// TIA Portal V20 export
FUNCTION_BLOCK "CallGlobal"   // FB48, LAD
TITLE = CallGlobal
// All blocks that provide data to the DB Global.Data are called here. That includes blocks to generate system data as well as blocks that connect handle multiple HMIs.
// stored: IsIECCheckEnabled true, MemoryReserve 100, SetENOAutomatically true
   VAR
      statClockSysMemOld { ExternalWritable := 'False'} : Byte;   // Old value system memory evaluation
      statRev0Hz5 : Bool;
      statTonTimer : Array[0..1] of IEC_TIMER;
      instLAF_PowerOnOff { ExternalWritable := 'False'} : "LAF_PowerOnOff";
      instLAF_HmiHeaderManager { ExternalWritable := 'False'} : "LAF_HmiHeaderManager";
      instLAF_ClockGen { ExternalWritable := 'False'} : "LAF_ClockGenerator";
      instLSNTP_Server { ExternalWritable := 'False'} : "LSNTP_Server";
      instRemoteAccess { ExternalWritable := 'False'} : "LRemoteAccess_MobilePanelMonitor";
      statPulse : Array[0..99] of Bool;
   END_VAR
   VAR_TEMP
      tempIndex : DInt;   // Temp variable for for loop
      tempAcknowledge : Bool;   // Summarized acknowledge command
      tempPowerOff : Bool;   // Summarized power off command
      tempPowerOn : Bool;   // Summarized power on command
      tempPowerStatus : Int;   // 0 - Off, 1 - Paused, 2 - On
      tempResultXor : Byte;   // Interim result of XOR operation
      tempPosPulse : Byte;   // Interim result puls calculation
   END_VAR
   VAR CONSTANT
      RESET_BUTTON__COULD_BE_ADDED_HERE : Bool := false;   // Placeholder for a potential global reset button
      TRUE : Bool := true;
      FALSE : Bool;
   END_VAR
   VAR_TEMP   // added for the SCL form of the ladder/FBD networks
      _w1 : Bool;
      _w2 : Bool;
      _w3 : Bool;
      _w4 : Bool;
   END_VAR
BEGIN

REGION Network 1 (SCL): Summarize HMI commands
   // Read commands for acknowledge, powerOn and powerOff from the different HMI panels and summarize them in temp variables for further logic in this block.
   // Initialize temp variables
   #tempAcknowledge :=
   #tempPowerOff :=
   #tempPowerOn := FALSE;

   // Loop through the HMI panels and summarize the commands
   FOR #tempIndex := 0 TO "NO_OF_PANELS" DO
       #tempAcknowledge := #tempAcknowledge OR "Hmi".mainHeader[#tempIndex].hmiToPlc.acknowledge;
       #tempPowerOff := #tempPowerOff OR "Hmi".mainHeader[#tempIndex].hmiToPlc.powerCommands.%X0;
       #tempPowerOn := #tempPowerOn OR "Hmi".mainHeader[#tempIndex].hmiToPlc.powerCommands.%X1;
   END_FOR;
END_REGION

REGION Network 2: Global Acknowledge
   // The global acknowledge command from the hmi button is assigned to Global.Data.general.acknowledge: This bit it forwarded to all underlaying modules
   // If a hard-wired global reset button exists, it can
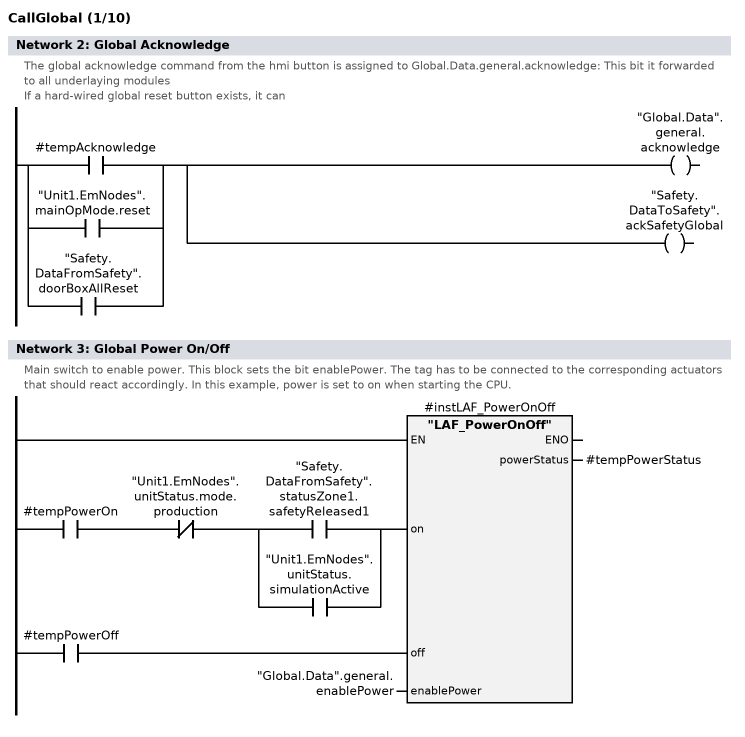
   RUNG wire#powerrail
      Contact( #tempAcknowledge )
      wire#w1
      Coil( "Global.Data".general.acknowledge )
   END_RUNG
   RUNG wire#powerrail
      Contact( "Unit1.EmNodes".mainOpMode.reset )
   END_RUNG wire#w1
   RUNG wire#powerrail
      Contact( "Safety.DataFromSafety".doorBoxAllReset )
   END_RUNG wire#w1
   RUNG wire#w1
      Coil( "Safety.DataToSafety".ackSafetyGlobal )
   END_RUNG
   // the same network as SCL:
   "Global.Data".general.acknowledge := #tempAcknowledge OR "Unit1.EmNodes".mainOpMode.reset OR "Safety.DataFromSafety".doorBoxAllReset;
   "Safety.DataToSafety".ackSafetyGlobal := "Global.Data".general.acknowledge;
END_REGION

REGION Network 3: Global Power On/Off
   // Main switch to enable power. This block sets the bit enablePower. The tag has to be connected to the corresponding actuators that should react accordingly. In this example, power is set to on when starting the CPU.
   RUNG wire#powerrail
      #instLAF_PowerOnOff(on := wire#w2, off := wire#w3, enablePower := "Global.Data".general.enablePower, powerStatus => #tempPowerStatus)
   END_RUNG
   RUNG wire#powerrail
      Contact( #tempPowerOn )
      I_Contact( "Unit1.EmNodes".unitStatus.mode.production )
      wire#w1
      Contact( "Safety.DataFromSafety".statusZone1.safetyReleased1 )
   END_RUNG wire#w2
   RUNG wire#w1
      Contact( "Unit1.EmNodes".unitStatus.simulationActive )
   END_RUNG wire#w2
   RUNG wire#powerrail
      Contact( #tempPowerOff )
   END_RUNG wire#w3
   // the same network as SCL:
   #instLAF_PowerOnOff(on := #tempPowerOn AND NOT "Unit1.EmNodes".unitStatus.mode.production AND ("Safety.DataFromSafety".statusZone1.safetyReleased1 OR "Unit1.EmNodes".unitStatus.simulationActive),   // "LAF_PowerOnOff"
                       off := #tempPowerOff,
                       enablePower := "Global.Data".general.enablePower,
                       powerStatus => #tempPowerStatus);
END_REGION

REGION Network 4 (SCL): Write power status to HMI panels
   // Write power status back to all connected HMI panels
   // Loop through the panels and set the power status
   FOR #tempIndex := 0 TO "NO_OF_PANELS" DO
       "Hmi".mainHeader[#tempIndex].plcToHmi.powerStatus := #tempPowerStatus;
   END_FOR;
END_REGION

REGION Network 5: Special Function Page1 Buttons l Operator Control Allowed
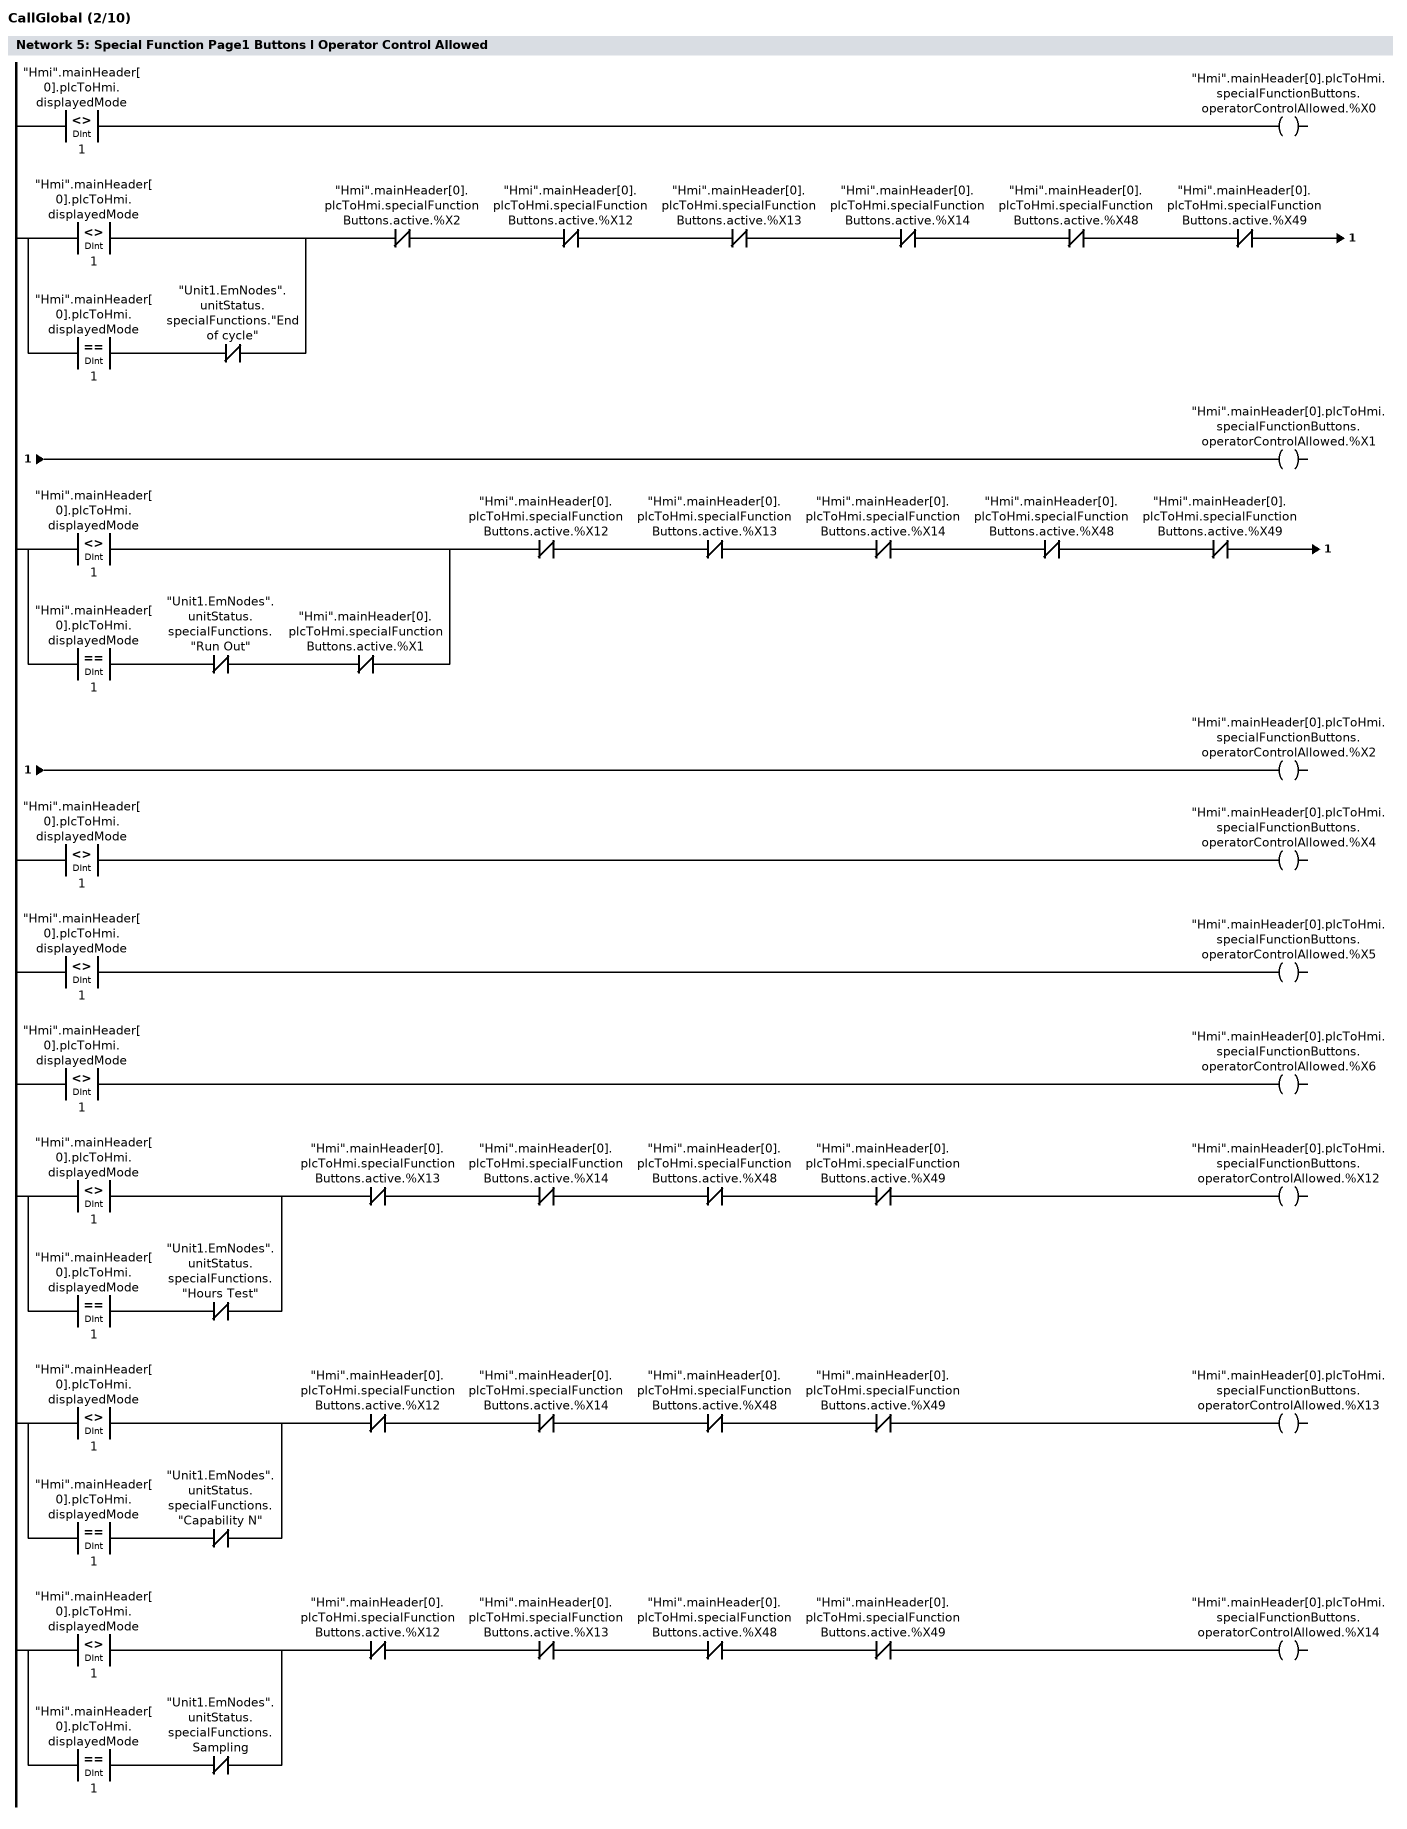
   RUNG wire#powerrail
      { S7_Templates := "SrcType := DInt" } NE_Contact(in1 := "Hmi".mainHeader[0].plcToHmi.displayedMode, in2 := 1)
      Coil( "Hmi".mainHeader[0].plcToHmi.specialFunctionButtons.operatorControlAllowed.%X0 )
   END_RUNG
   RUNG wire#powerrail
      { S7_Templates := "SrcType := DInt" } NE_Contact(in1 := "Hmi".mainHeader[0].plcToHmi.displayedMode, in2 := 1)
      wire#w1
      I_Contact( "Hmi".mainHeader[0].plcToHmi.specialFunctionButtons.active.%X2 )
      I_Contact( "Hmi".mainHeader[0].plcToHmi.specialFunctionButtons.active.%X12 )
      I_Contact( "Hmi".mainHeader[0].plcToHmi.specialFunctionButtons.active.%X13 )
      I_Contact( "Hmi".mainHeader[0].plcToHmi.specialFunctionButtons.active.%X14 )
      I_Contact( "Hmi".mainHeader[0].plcToHmi.specialFunctionButtons.active.%X48 )
      I_Contact( "Hmi".mainHeader[0].plcToHmi.specialFunctionButtons.active.%X49 )
      Coil( "Hmi".mainHeader[0].plcToHmi.specialFunctionButtons.operatorControlAllowed.%X1 )
   END_RUNG
   RUNG wire#powerrail
      { S7_Templates := "SrcType := DInt" } EQ_Contact(in1 := "Hmi".mainHeader[0].plcToHmi.displayedMode, in2 := 1)
      I_Contact( "Unit1.EmNodes".unitStatus.specialFunctions."End of cycle" )
   END_RUNG wire#w1
   RUNG wire#powerrail
      { S7_Templates := "SrcType := DInt" } NE_Contact(in1 := "Hmi".mainHeader[0].plcToHmi.displayedMode, in2 := 1)
      wire#w2
      I_Contact( "Hmi".mainHeader[0].plcToHmi.specialFunctionButtons.active.%X12 )
      I_Contact( "Hmi".mainHeader[0].plcToHmi.specialFunctionButtons.active.%X13 )
      I_Contact( "Hmi".mainHeader[0].plcToHmi.specialFunctionButtons.active.%X14 )
      I_Contact( "Hmi".mainHeader[0].plcToHmi.specialFunctionButtons.active.%X48 )
      I_Contact( "Hmi".mainHeader[0].plcToHmi.specialFunctionButtons.active.%X49 )
      Coil( "Hmi".mainHeader[0].plcToHmi.specialFunctionButtons.operatorControlAllowed.%X2 )
   END_RUNG
   RUNG wire#powerrail
      { S7_Templates := "SrcType := DInt" } EQ_Contact(in1 := "Hmi".mainHeader[0].plcToHmi.displayedMode, in2 := 1)
      I_Contact( "Unit1.EmNodes".unitStatus.specialFunctions."Run Out" )
      I_Contact( "Hmi".mainHeader[0].plcToHmi.specialFunctionButtons.active.%X1 )
   END_RUNG wire#w2
   RUNG wire#powerrail
      { S7_Templates := "SrcType := DInt" } NE_Contact(in1 := "Hmi".mainHeader[0].plcToHmi.displayedMode, in2 := 1)
      Coil( "Hmi".mainHeader[0].plcToHmi.specialFunctionButtons.operatorControlAllowed.%X4 )
   END_RUNG
   RUNG wire#powerrail
      { S7_Templates := "SrcType := DInt" } NE_Contact(in1 := "Hmi".mainHeader[0].plcToHmi.displayedMode, in2 := 1)
      Coil( "Hmi".mainHeader[0].plcToHmi.specialFunctionButtons.operatorControlAllowed.%X5 )
   END_RUNG
   RUNG wire#powerrail
      { S7_Templates := "SrcType := DInt" } NE_Contact(in1 := "Hmi".mainHeader[0].plcToHmi.displayedMode, in2 := 1)
      Coil( "Hmi".mainHeader[0].plcToHmi.specialFunctionButtons.operatorControlAllowed.%X6 )
   END_RUNG
   RUNG wire#powerrail
      { S7_Templates := "SrcType := DInt" } NE_Contact(in1 := "Hmi".mainHeader[0].plcToHmi.displayedMode, in2 := 1)
      wire#w3
      I_Contact( "Hmi".mainHeader[0].plcToHmi.specialFunctionButtons.active.%X13 )
      I_Contact( "Hmi".mainHeader[0].plcToHmi.specialFunctionButtons.active.%X14 )
      I_Contact( "Hmi".mainHeader[0].plcToHmi.specialFunctionButtons.active.%X48 )
      I_Contact( "Hmi".mainHeader[0].plcToHmi.specialFunctionButtons.active.%X49 )
      Coil( "Hmi".mainHeader[0].plcToHmi.specialFunctionButtons.operatorControlAllowed.%X12 )
   END_RUNG
   RUNG wire#powerrail
      { S7_Templates := "SrcType := DInt" } EQ_Contact(in1 := "Hmi".mainHeader[0].plcToHmi.displayedMode, in2 := 1)
      I_Contact( "Unit1.EmNodes".unitStatus.specialFunctions."Hours Test" )
   END_RUNG wire#w3
   RUNG wire#powerrail
      { S7_Templates := "SrcType := DInt" } NE_Contact(in1 := "Hmi".mainHeader[0].plcToHmi.displayedMode, in2 := 1)
      wire#w4
      I_Contact( "Hmi".mainHeader[0].plcToHmi.specialFunctionButtons.active.%X12 )
      I_Contact( "Hmi".mainHeader[0].plcToHmi.specialFunctionButtons.active.%X14 )
      I_Contact( "Hmi".mainHeader[0].plcToHmi.specialFunctionButtons.active.%X48 )
      I_Contact( "Hmi".mainHeader[0].plcToHmi.specialFunctionButtons.active.%X49 )
      Coil( "Hmi".mainHeader[0].plcToHmi.specialFunctionButtons.operatorControlAllowed.%X13 )
   END_RUNG
   RUNG wire#powerrail
      { S7_Templates := "SrcType := DInt" } EQ_Contact(in1 := "Hmi".mainHeader[0].plcToHmi.displayedMode, in2 := 1)
      I_Contact( "Unit1.EmNodes".unitStatus.specialFunctions."Capability N" )
   END_RUNG wire#w4
   RUNG wire#powerrail
      { S7_Templates := "SrcType := DInt" } NE_Contact(in1 := "Hmi".mainHeader[0].plcToHmi.displayedMode, in2 := 1)
      wire#w5
      I_Contact( "Hmi".mainHeader[0].plcToHmi.specialFunctionButtons.active.%X12 )
      I_Contact( "Hmi".mainHeader[0].plcToHmi.specialFunctionButtons.active.%X13 )
      I_Contact( "Hmi".mainHeader[0].plcToHmi.specialFunctionButtons.active.%X48 )
      I_Contact( "Hmi".mainHeader[0].plcToHmi.specialFunctionButtons.active.%X49 )
      Coil( "Hmi".mainHeader[0].plcToHmi.specialFunctionButtons.operatorControlAllowed.%X14 )
   END_RUNG
   RUNG wire#powerrail
      { S7_Templates := "SrcType := DInt" } EQ_Contact(in1 := "Hmi".mainHeader[0].plcToHmi.displayedMode, in2 := 1)
      I_Contact( "Unit1.EmNodes".unitStatus.specialFunctions.Sampling )
   END_RUNG wire#w5
   // the same network as SCL:
   "Hmi".mainHeader[0].plcToHmi.specialFunctionButtons.operatorControlAllowed.%X0 := "Hmi".mainHeader[0].plcToHmi.displayedMode <> 1;
   "Hmi".mainHeader[0].plcToHmi.specialFunctionButtons.operatorControlAllowed.%X1 := (("Hmi".mainHeader[0].plcToHmi.displayedMode <> 1) OR (("Hmi".mainHeader[0].plcToHmi.displayedMode = 1) AND NOT "Unit1.EmNodes".unitStatus.specialFunctions."End of cycle")) AND NOT "Hmi".mainHeader[0].plcToHmi.specialFunctionButtons.active.%X2 AND NOT "Hmi".mainHeader[0].plcToHmi.specialFunctionButtons.active.%X12 AND NOT "Hmi".mainHeader[0].plcToHmi.specialFunctionButtons.active.%X13 AND NOT "Hmi".mainHeader[0].plcToHmi.specialFunctionButtons.active.%X14 AND NOT "Hmi".mainHeader[0].plcToHmi.specialFunctionButtons.active.%X48 AND NOT "Hmi".mainHeader[0].plcToHmi.specialFunctionButtons.active.%X49;
   "Hmi".mainHeader[0].plcToHmi.specialFunctionButtons.operatorControlAllowed.%X2 := (("Hmi".mainHeader[0].plcToHmi.displayedMode <> 1) OR (("Hmi".mainHeader[0].plcToHmi.displayedMode = 1) AND NOT "Unit1.EmNodes".unitStatus.specialFunctions."Run Out" AND NOT "Hmi".mainHeader[0].plcToHmi.specialFunctionButtons.active.%X1)) AND NOT "Hmi".mainHeader[0].plcToHmi.specialFunctionButtons.active.%X12 AND NOT "Hmi".mainHeader[0].plcToHmi.specialFunctionButtons.active.%X13 AND NOT "Hmi".mainHeader[0].plcToHmi.specialFunctionButtons.active.%X14 AND NOT "Hmi".mainHeader[0].plcToHmi.specialFunctionButtons.active.%X48 AND NOT "Hmi".mainHeader[0].plcToHmi.specialFunctionButtons.active.%X49;
   "Hmi".mainHeader[0].plcToHmi.specialFunctionButtons.operatorControlAllowed.%X4 := "Hmi".mainHeader[0].plcToHmi.displayedMode <> 1;
   "Hmi".mainHeader[0].plcToHmi.specialFunctionButtons.operatorControlAllowed.%X5 := "Hmi".mainHeader[0].plcToHmi.displayedMode <> 1;
   "Hmi".mainHeader[0].plcToHmi.specialFunctionButtons.operatorControlAllowed.%X6 := "Hmi".mainHeader[0].plcToHmi.displayedMode <> 1;
   "Hmi".mainHeader[0].plcToHmi.specialFunctionButtons.operatorControlAllowed.%X12 := (("Hmi".mainHeader[0].plcToHmi.displayedMode <> 1) OR (("Hmi".mainHeader[0].plcToHmi.displayedMode = 1) AND NOT "Unit1.EmNodes".unitStatus.specialFunctions."Hours Test")) AND NOT "Hmi".mainHeader[0].plcToHmi.specialFunctionButtons.active.%X13 AND NOT "Hmi".mainHeader[0].plcToHmi.specialFunctionButtons.active.%X14 AND NOT "Hmi".mainHeader[0].plcToHmi.specialFunctionButtons.active.%X48 AND NOT "Hmi".mainHeader[0].plcToHmi.specialFunctionButtons.active.%X49;
   "Hmi".mainHeader[0].plcToHmi.specialFunctionButtons.operatorControlAllowed.%X13 := (("Hmi".mainHeader[0].plcToHmi.displayedMode <> 1) OR (("Hmi".mainHeader[0].plcToHmi.displayedMode = 1) AND NOT "Unit1.EmNodes".unitStatus.specialFunctions."Capability N")) AND NOT "Hmi".mainHeader[0].plcToHmi.specialFunctionButtons.active.%X12 AND NOT "Hmi".mainHeader[0].plcToHmi.specialFunctionButtons.active.%X14 AND NOT "Hmi".mainHeader[0].plcToHmi.specialFunctionButtons.active.%X48 AND NOT "Hmi".mainHeader[0].plcToHmi.specialFunctionButtons.active.%X49;
   "Hmi".mainHeader[0].plcToHmi.specialFunctionButtons.operatorControlAllowed.%X14 := (("Hmi".mainHeader[0].plcToHmi.displayedMode <> 1) OR (("Hmi".mainHeader[0].plcToHmi.displayedMode = 1) AND NOT "Unit1.EmNodes".unitStatus.specialFunctions.Sampling)) AND NOT "Hmi".mainHeader[0].plcToHmi.specialFunctionButtons.active.%X12 AND NOT "Hmi".mainHeader[0].plcToHmi.specialFunctionButtons.active.%X13 AND NOT "Hmi".mainHeader[0].plcToHmi.specialFunctionButtons.active.%X48 AND NOT "Hmi".mainHeader[0].plcToHmi.specialFunctionButtons.active.%X49;
END_REGION

REGION Network 6: Special Function Page2 Buttons l Operator Control Allowed
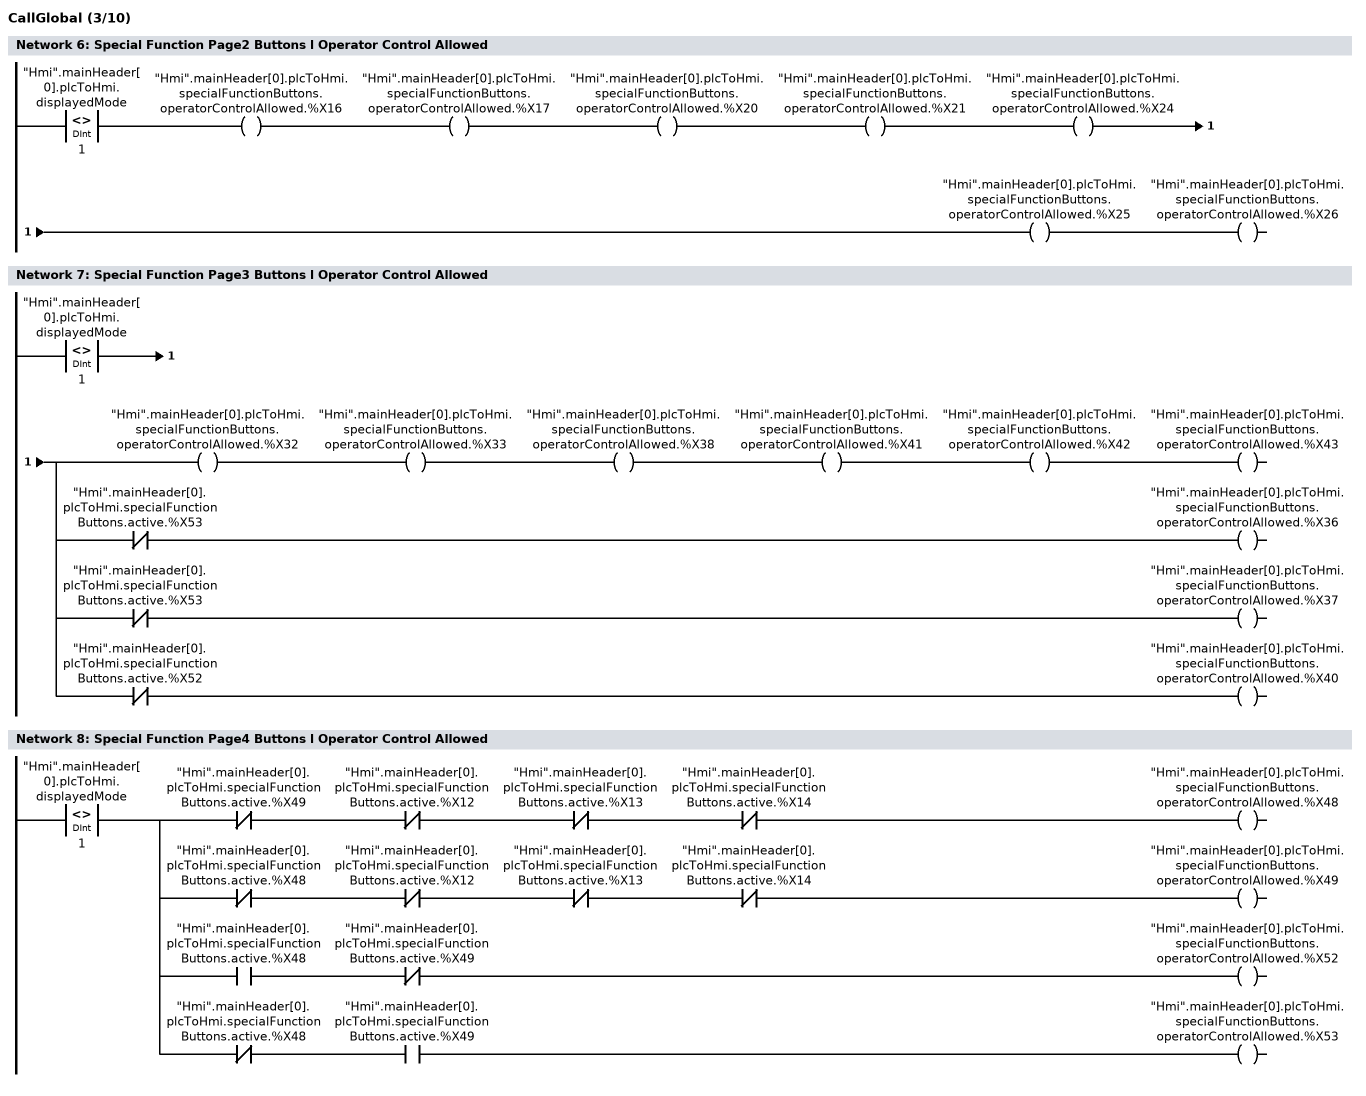
   RUNG wire#powerrail
      { S7_Templates := "SrcType := DInt" } NE_Contact(in1 := "Hmi".mainHeader[0].plcToHmi.displayedMode, in2 := 1)
      Coil( "Hmi".mainHeader[0].plcToHmi.specialFunctionButtons.operatorControlAllowed.%X16 )
      Coil( "Hmi".mainHeader[0].plcToHmi.specialFunctionButtons.operatorControlAllowed.%X17 )
      Coil( "Hmi".mainHeader[0].plcToHmi.specialFunctionButtons.operatorControlAllowed.%X20 )
      Coil( "Hmi".mainHeader[0].plcToHmi.specialFunctionButtons.operatorControlAllowed.%X21 )
      Coil( "Hmi".mainHeader[0].plcToHmi.specialFunctionButtons.operatorControlAllowed.%X24 )
      Coil( "Hmi".mainHeader[0].plcToHmi.specialFunctionButtons.operatorControlAllowed.%X25 )
      Coil( "Hmi".mainHeader[0].plcToHmi.specialFunctionButtons.operatorControlAllowed.%X26 )
   END_RUNG
   // the same network as SCL:
   #_w1 := "Hmi".mainHeader[0].plcToHmi.displayedMode <> 1;
   "Hmi".mainHeader[0].plcToHmi.specialFunctionButtons.operatorControlAllowed.%X16 := #_w1;
   "Hmi".mainHeader[0].plcToHmi.specialFunctionButtons.operatorControlAllowed.%X17 := #_w1;
   "Hmi".mainHeader[0].plcToHmi.specialFunctionButtons.operatorControlAllowed.%X20 := #_w1;
   "Hmi".mainHeader[0].plcToHmi.specialFunctionButtons.operatorControlAllowed.%X21 := #_w1;
   "Hmi".mainHeader[0].plcToHmi.specialFunctionButtons.operatorControlAllowed.%X24 := #_w1;
   "Hmi".mainHeader[0].plcToHmi.specialFunctionButtons.operatorControlAllowed.%X25 := #_w1;
   "Hmi".mainHeader[0].plcToHmi.specialFunctionButtons.operatorControlAllowed.%X26 := #_w1;
END_REGION

REGION Network 7: Special Function Page3 Buttons l Operator Control Allowed
   RUNG wire#powerrail
      { S7_Templates := "SrcType := DInt" } NE_Contact(in1 := "Hmi".mainHeader[0].plcToHmi.displayedMode, in2 := 1)
      wire#w1
      Coil( "Hmi".mainHeader[0].plcToHmi.specialFunctionButtons.operatorControlAllowed.%X32 )
      Coil( "Hmi".mainHeader[0].plcToHmi.specialFunctionButtons.operatorControlAllowed.%X33 )
      Coil( "Hmi".mainHeader[0].plcToHmi.specialFunctionButtons.operatorControlAllowed.%X38 )
      Coil( "Hmi".mainHeader[0].plcToHmi.specialFunctionButtons.operatorControlAllowed.%X41 )
      Coil( "Hmi".mainHeader[0].plcToHmi.specialFunctionButtons.operatorControlAllowed.%X42 )
      Coil( "Hmi".mainHeader[0].plcToHmi.specialFunctionButtons.operatorControlAllowed.%X43 )
   END_RUNG
   RUNG wire#w1
      I_Contact( "Hmi".mainHeader[0].plcToHmi.specialFunctionButtons.active.%X53 )
      Coil( "Hmi".mainHeader[0].plcToHmi.specialFunctionButtons.operatorControlAllowed.%X36 )
   END_RUNG
   RUNG wire#w1
      I_Contact( "Hmi".mainHeader[0].plcToHmi.specialFunctionButtons.active.%X53 )
      Coil( "Hmi".mainHeader[0].plcToHmi.specialFunctionButtons.operatorControlAllowed.%X37 )
   END_RUNG
   RUNG wire#w1
      I_Contact( "Hmi".mainHeader[0].plcToHmi.specialFunctionButtons.active.%X52 )
      Coil( "Hmi".mainHeader[0].plcToHmi.specialFunctionButtons.operatorControlAllowed.%X40 )
   END_RUNG
   // the same network as SCL:
   #_w1 := "Hmi".mainHeader[0].plcToHmi.displayedMode <> 1;
   "Hmi".mainHeader[0].plcToHmi.specialFunctionButtons.operatorControlAllowed.%X32 := #_w1;
   "Hmi".mainHeader[0].plcToHmi.specialFunctionButtons.operatorControlAllowed.%X33 := #_w1;
   "Hmi".mainHeader[0].plcToHmi.specialFunctionButtons.operatorControlAllowed.%X38 := #_w1;
   "Hmi".mainHeader[0].plcToHmi.specialFunctionButtons.operatorControlAllowed.%X41 := #_w1;
   "Hmi".mainHeader[0].plcToHmi.specialFunctionButtons.operatorControlAllowed.%X42 := #_w1;
   "Hmi".mainHeader[0].plcToHmi.specialFunctionButtons.operatorControlAllowed.%X43 := #_w1;
   "Hmi".mainHeader[0].plcToHmi.specialFunctionButtons.operatorControlAllowed.%X36 := #_w1 AND NOT "Hmi".mainHeader[0].plcToHmi.specialFunctionButtons.active.%X53;
   "Hmi".mainHeader[0].plcToHmi.specialFunctionButtons.operatorControlAllowed.%X37 := #_w1 AND NOT "Hmi".mainHeader[0].plcToHmi.specialFunctionButtons.active.%X53;
   "Hmi".mainHeader[0].plcToHmi.specialFunctionButtons.operatorControlAllowed.%X40 := #_w1 AND NOT "Hmi".mainHeader[0].plcToHmi.specialFunctionButtons.active.%X52;
END_REGION

REGION Network 8: Special Function Page4 Buttons l Operator Control Allowed
   RUNG wire#powerrail
      { S7_Templates := "SrcType := DInt" } NE_Contact(in1 := "Hmi".mainHeader[0].plcToHmi.displayedMode, in2 := 1)
      wire#w1
      I_Contact( "Hmi".mainHeader[0].plcToHmi.specialFunctionButtons.active.%X49 )
      I_Contact( "Hmi".mainHeader[0].plcToHmi.specialFunctionButtons.active.%X12 )
      I_Contact( "Hmi".mainHeader[0].plcToHmi.specialFunctionButtons.active.%X13 )
      I_Contact( "Hmi".mainHeader[0].plcToHmi.specialFunctionButtons.active.%X14 )
      Coil( "Hmi".mainHeader[0].plcToHmi.specialFunctionButtons.operatorControlAllowed.%X48 )
   END_RUNG
   RUNG wire#w1
      I_Contact( "Hmi".mainHeader[0].plcToHmi.specialFunctionButtons.active.%X48 )
      I_Contact( "Hmi".mainHeader[0].plcToHmi.specialFunctionButtons.active.%X12 )
      I_Contact( "Hmi".mainHeader[0].plcToHmi.specialFunctionButtons.active.%X13 )
      I_Contact( "Hmi".mainHeader[0].plcToHmi.specialFunctionButtons.active.%X14 )
      Coil( "Hmi".mainHeader[0].plcToHmi.specialFunctionButtons.operatorControlAllowed.%X49 )
   END_RUNG
   RUNG wire#w1
      Contact( "Hmi".mainHeader[0].plcToHmi.specialFunctionButtons.active.%X48 )
      I_Contact( "Hmi".mainHeader[0].plcToHmi.specialFunctionButtons.active.%X49 )
      Coil( "Hmi".mainHeader[0].plcToHmi.specialFunctionButtons.operatorControlAllowed.%X52 )
   END_RUNG
   RUNG wire#w1
      I_Contact( "Hmi".mainHeader[0].plcToHmi.specialFunctionButtons.active.%X48 )
      Contact( "Hmi".mainHeader[0].plcToHmi.specialFunctionButtons.active.%X49 )
      Coil( "Hmi".mainHeader[0].plcToHmi.specialFunctionButtons.operatorControlAllowed.%X53 )
   END_RUNG
   // the same network as SCL:
   #_w1 := "Hmi".mainHeader[0].plcToHmi.displayedMode <> 1;
   "Hmi".mainHeader[0].plcToHmi.specialFunctionButtons.operatorControlAllowed.%X48 := #_w1 AND NOT "Hmi".mainHeader[0].plcToHmi.specialFunctionButtons.active.%X49 AND NOT "Hmi".mainHeader[0].plcToHmi.specialFunctionButtons.active.%X12 AND NOT "Hmi".mainHeader[0].plcToHmi.specialFunctionButtons.active.%X13 AND NOT "Hmi".mainHeader[0].plcToHmi.specialFunctionButtons.active.%X14;
   "Hmi".mainHeader[0].plcToHmi.specialFunctionButtons.operatorControlAllowed.%X49 := #_w1 AND NOT "Hmi".mainHeader[0].plcToHmi.specialFunctionButtons.active.%X48 AND NOT "Hmi".mainHeader[0].plcToHmi.specialFunctionButtons.active.%X12 AND NOT "Hmi".mainHeader[0].plcToHmi.specialFunctionButtons.active.%X13 AND NOT "Hmi".mainHeader[0].plcToHmi.specialFunctionButtons.active.%X14;
   "Hmi".mainHeader[0].plcToHmi.specialFunctionButtons.operatorControlAllowed.%X52 := #_w1 AND "Hmi".mainHeader[0].plcToHmi.specialFunctionButtons.active.%X48 AND NOT "Hmi".mainHeader[0].plcToHmi.specialFunctionButtons.active.%X49;
   "Hmi".mainHeader[0].plcToHmi.specialFunctionButtons.operatorControlAllowed.%X53 := #_w1 AND NOT "Hmi".mainHeader[0].plcToHmi.specialFunctionButtons.active.%X48 AND "Hmi".mainHeader[0].plcToHmi.specialFunctionButtons.active.%X49;
END_REGION

REGION Network 9: Special Function Buttons l Gauge R&R Type1
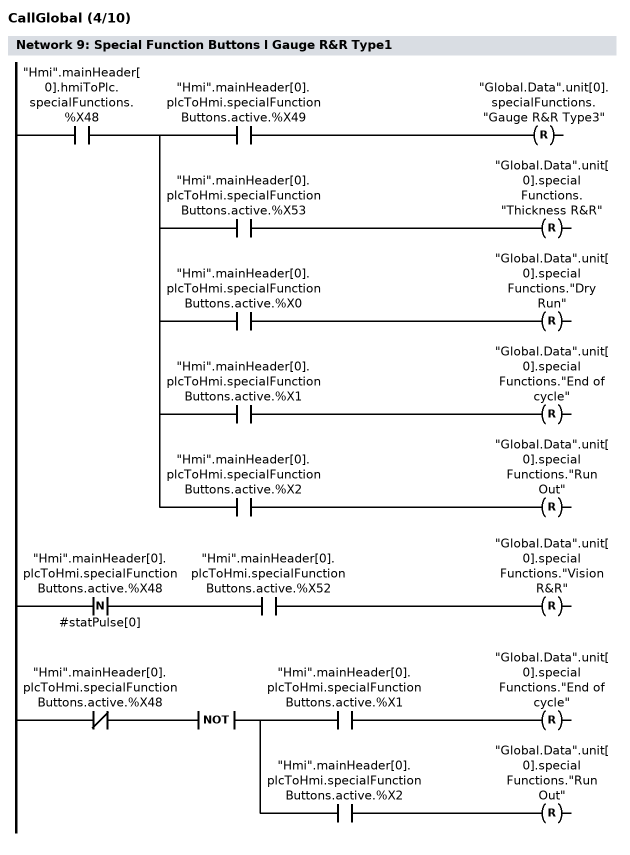
   RUNG wire#powerrail
      Contact( "Hmi".mainHeader[0].hmiToPlc.specialFunctions.%X48 )
      wire#w1
      Contact( "Hmi".mainHeader[0].plcToHmi.specialFunctionButtons.active.%X49 )
      R_Coil( "Global.Data".unit[0].specialFunctions."Gauge R&R Type3" )
   END_RUNG
   RUNG wire#w1
      Contact( "Hmi".mainHeader[0].plcToHmi.specialFunctionButtons.active.%X53 )
      R_Coil( "Global.Data".unit[0].specialFunctions."Thickness R&R" )
   END_RUNG
   RUNG wire#w1
      Contact( "Hmi".mainHeader[0].plcToHmi.specialFunctionButtons.active.%X0 )
      R_Coil( "Global.Data".unit[0].specialFunctions."Dry Run" )
   END_RUNG
   RUNG wire#w1
      Contact( "Hmi".mainHeader[0].plcToHmi.specialFunctionButtons.active.%X1 )
      R_Coil( "Global.Data".unit[0].specialFunctions."End of cycle" )
   END_RUNG
   RUNG wire#w1
      Contact( "Hmi".mainHeader[0].plcToHmi.specialFunctionButtons.active.%X2 )
      R_Coil( "Global.Data".unit[0].specialFunctions."Run Out" )
   END_RUNG
   RUNG wire#powerrail
      N_Contact(operand := "Hmi".mainHeader[0].plcToHmi.specialFunctionButtons.active.%X48, bit := #statPulse[0])
      Contact( "Hmi".mainHeader[0].plcToHmi.specialFunctionButtons.active.%X52 )
      R_Coil( "Global.Data".unit[0].specialFunctions."Vision R&R" )
   END_RUNG
   RUNG wire#powerrail
      I_Contact( "Hmi".mainHeader[0].plcToHmi.specialFunctionButtons.active.%X48 )
      Not()
      wire#w2
      Contact( "Hmi".mainHeader[0].plcToHmi.specialFunctionButtons.active.%X1 )
      R_Coil( "Global.Data".unit[0].specialFunctions."End of cycle" )
   END_RUNG
   RUNG wire#w2
      Contact( "Hmi".mainHeader[0].plcToHmi.specialFunctionButtons.active.%X2 )
      R_Coil( "Global.Data".unit[0].specialFunctions."Run Out" )
   END_RUNG
   // the same network as SCL:
   IF "Hmi".mainHeader[0].hmiToPlc.specialFunctions.%X48 AND "Hmi".mainHeader[0].plcToHmi.specialFunctionButtons.active.%X49 THEN
       "Global.Data".unit[0].specialFunctions."Gauge R&R Type3" := FALSE;
   END_IF;
   IF "Hmi".mainHeader[0].hmiToPlc.specialFunctions.%X48 AND "Hmi".mainHeader[0].plcToHmi.specialFunctionButtons.active.%X53 THEN
       "Global.Data".unit[0].specialFunctions."Thickness R&R" := FALSE;
   END_IF;
   IF "Hmi".mainHeader[0].hmiToPlc.specialFunctions.%X48 AND "Hmi".mainHeader[0].plcToHmi.specialFunctionButtons.active.%X0 THEN
       "Global.Data".unit[0].specialFunctions."Dry Run" := FALSE;
   END_IF;
   IF "Hmi".mainHeader[0].hmiToPlc.specialFunctions.%X48 AND "Hmi".mainHeader[0].plcToHmi.specialFunctionButtons.active.%X1 THEN
       "Global.Data".unit[0].specialFunctions."End of cycle" := FALSE;
   END_IF;
   IF "Hmi".mainHeader[0].hmiToPlc.specialFunctions.%X48 AND "Hmi".mainHeader[0].plcToHmi.specialFunctionButtons.active.%X2 THEN
       "Global.Data".unit[0].specialFunctions."Run Out" := FALSE;
   END_IF;
   #_w1 := NOT "Hmi".mainHeader[0].plcToHmi.specialFunctionButtons.active.%X48 AND #statPulse[0];   // falling edge of "Hmi".mainHeader[0].plcToHmi.specialFunctionButtons.active.%X48
   #statPulse[0] := "Hmi".mainHeader[0].plcToHmi.specialFunctionButtons.active.%X48;
   IF #_w1 AND "Hmi".mainHeader[0].plcToHmi.specialFunctionButtons.active.%X52 THEN
       "Global.Data".unit[0].specialFunctions."Vision R&R" := FALSE;
   END_IF;
   #_w2 := NOT (NOT "Hmi".mainHeader[0].plcToHmi.specialFunctionButtons.active.%X48);
   IF #_w2 AND "Hmi".mainHeader[0].plcToHmi.specialFunctionButtons.active.%X1 THEN
       "Global.Data".unit[0].specialFunctions."End of cycle" := FALSE;
   END_IF;
   IF #_w2 AND "Hmi".mainHeader[0].plcToHmi.specialFunctionButtons.active.%X2 THEN
       "Global.Data".unit[0].specialFunctions."Run Out" := FALSE;
   END_IF;
END_REGION

REGION Network 10: Special Function Buttons l Gauge R&R Type3
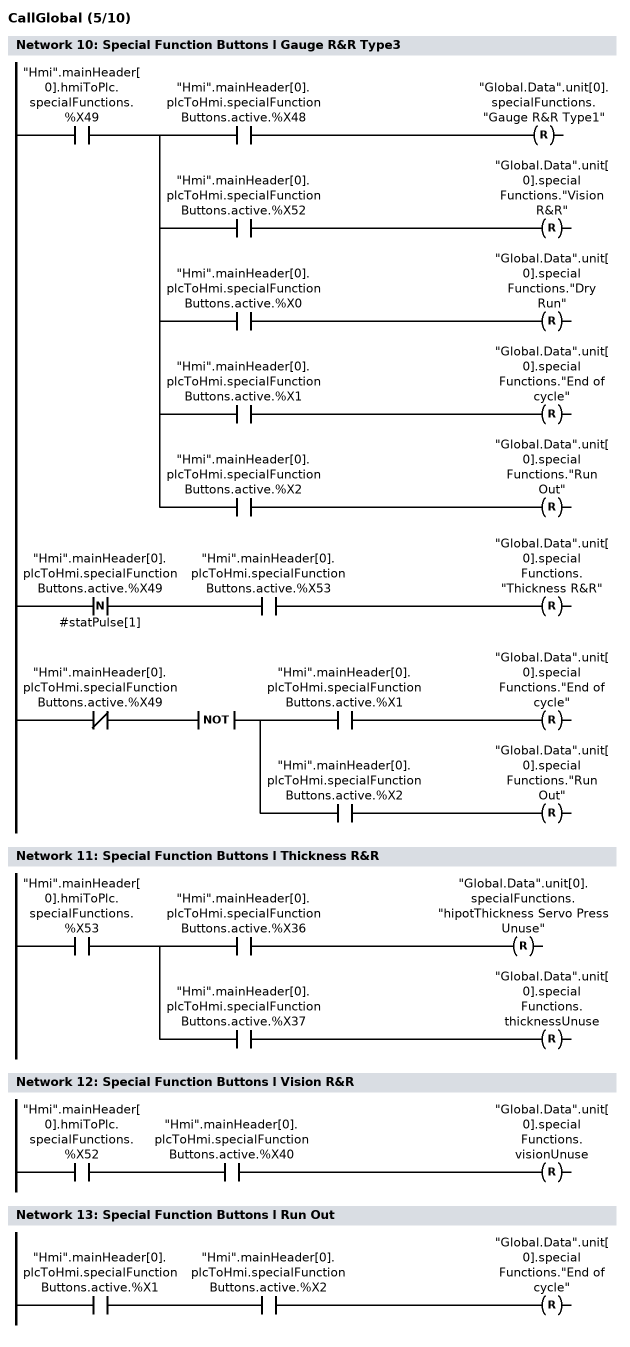
   RUNG wire#powerrail
      Contact( "Hmi".mainHeader[0].hmiToPlc.specialFunctions.%X49 )
      wire#w1
      Contact( "Hmi".mainHeader[0].plcToHmi.specialFunctionButtons.active.%X48 )
      R_Coil( "Global.Data".unit[0].specialFunctions."Gauge R&R Type1" )
   END_RUNG
   RUNG wire#w1
      Contact( "Hmi".mainHeader[0].plcToHmi.specialFunctionButtons.active.%X52 )
      R_Coil( "Global.Data".unit[0].specialFunctions."Vision R&R" )
   END_RUNG
   RUNG wire#w1
      Contact( "Hmi".mainHeader[0].plcToHmi.specialFunctionButtons.active.%X0 )
      R_Coil( "Global.Data".unit[0].specialFunctions."Dry Run" )
   END_RUNG
   RUNG wire#w1
      Contact( "Hmi".mainHeader[0].plcToHmi.specialFunctionButtons.active.%X1 )
      R_Coil( "Global.Data".unit[0].specialFunctions."End of cycle" )
   END_RUNG
   RUNG wire#w1
      Contact( "Hmi".mainHeader[0].plcToHmi.specialFunctionButtons.active.%X2 )
      R_Coil( "Global.Data".unit[0].specialFunctions."Run Out" )
   END_RUNG
   RUNG wire#powerrail
      N_Contact(operand := "Hmi".mainHeader[0].plcToHmi.specialFunctionButtons.active.%X49, bit := #statPulse[1])
      Contact( "Hmi".mainHeader[0].plcToHmi.specialFunctionButtons.active.%X53 )
      R_Coil( "Global.Data".unit[0].specialFunctions."Thickness R&R" )
   END_RUNG
   RUNG wire#powerrail
      I_Contact( "Hmi".mainHeader[0].plcToHmi.specialFunctionButtons.active.%X49 )
      Not()
      wire#w2
      Contact( "Hmi".mainHeader[0].plcToHmi.specialFunctionButtons.active.%X1 )
      R_Coil( "Global.Data".unit[0].specialFunctions."End of cycle" )
   END_RUNG
   RUNG wire#w2
      Contact( "Hmi".mainHeader[0].plcToHmi.specialFunctionButtons.active.%X2 )
      R_Coil( "Global.Data".unit[0].specialFunctions."Run Out" )
   END_RUNG
   // the same network as SCL:
   IF "Hmi".mainHeader[0].hmiToPlc.specialFunctions.%X49 AND "Hmi".mainHeader[0].plcToHmi.specialFunctionButtons.active.%X48 THEN
       "Global.Data".unit[0].specialFunctions."Gauge R&R Type1" := FALSE;
   END_IF;
   IF "Hmi".mainHeader[0].hmiToPlc.specialFunctions.%X49 AND "Hmi".mainHeader[0].plcToHmi.specialFunctionButtons.active.%X52 THEN
       "Global.Data".unit[0].specialFunctions."Vision R&R" := FALSE;
   END_IF;
   IF "Hmi".mainHeader[0].hmiToPlc.specialFunctions.%X49 AND "Hmi".mainHeader[0].plcToHmi.specialFunctionButtons.active.%X0 THEN
       "Global.Data".unit[0].specialFunctions."Dry Run" := FALSE;
   END_IF;
   IF "Hmi".mainHeader[0].hmiToPlc.specialFunctions.%X49 AND "Hmi".mainHeader[0].plcToHmi.specialFunctionButtons.active.%X1 THEN
       "Global.Data".unit[0].specialFunctions."End of cycle" := FALSE;
   END_IF;
   IF "Hmi".mainHeader[0].hmiToPlc.specialFunctions.%X49 AND "Hmi".mainHeader[0].plcToHmi.specialFunctionButtons.active.%X2 THEN
       "Global.Data".unit[0].specialFunctions."Run Out" := FALSE;
   END_IF;
   #_w1 := NOT "Hmi".mainHeader[0].plcToHmi.specialFunctionButtons.active.%X49 AND #statPulse[1];   // falling edge of "Hmi".mainHeader[0].plcToHmi.specialFunctionButtons.active.%X49
   #statPulse[1] := "Hmi".mainHeader[0].plcToHmi.specialFunctionButtons.active.%X49;
   IF #_w1 AND "Hmi".mainHeader[0].plcToHmi.specialFunctionButtons.active.%X53 THEN
       "Global.Data".unit[0].specialFunctions."Thickness R&R" := FALSE;
   END_IF;
   #_w2 := NOT (NOT "Hmi".mainHeader[0].plcToHmi.specialFunctionButtons.active.%X49);
   IF #_w2 AND "Hmi".mainHeader[0].plcToHmi.specialFunctionButtons.active.%X1 THEN
       "Global.Data".unit[0].specialFunctions."End of cycle" := FALSE;
   END_IF;
   IF #_w2 AND "Hmi".mainHeader[0].plcToHmi.specialFunctionButtons.active.%X2 THEN
       "Global.Data".unit[0].specialFunctions."Run Out" := FALSE;
   END_IF;
END_REGION

REGION Network 11: Special Function Buttons l Thickness R&R
   RUNG wire#powerrail
      Contact( "Hmi".mainHeader[0].hmiToPlc.specialFunctions.%X53 )
      wire#w1
      Contact( "Hmi".mainHeader[0].plcToHmi.specialFunctionButtons.active.%X36 )
      R_Coil( "Global.Data".unit[0].specialFunctions."hipotThickness Servo Press Unuse" )
   END_RUNG
   RUNG wire#w1
      Contact( "Hmi".mainHeader[0].plcToHmi.specialFunctionButtons.active.%X37 )
      R_Coil( "Global.Data".unit[0].specialFunctions.thicknessUnuse )
   END_RUNG
   // the same network as SCL:
   IF "Hmi".mainHeader[0].hmiToPlc.specialFunctions.%X53 AND "Hmi".mainHeader[0].plcToHmi.specialFunctionButtons.active.%X36 THEN
       "Global.Data".unit[0].specialFunctions."hipotThickness Servo Press Unuse" := FALSE;
   END_IF;
   IF "Hmi".mainHeader[0].hmiToPlc.specialFunctions.%X53 AND "Hmi".mainHeader[0].plcToHmi.specialFunctionButtons.active.%X37 THEN
       "Global.Data".unit[0].specialFunctions.thicknessUnuse := FALSE;
   END_IF;
END_REGION

REGION Network 12: Special Function Buttons l Vision R&R
   RUNG wire#powerrail
      Contact( "Hmi".mainHeader[0].hmiToPlc.specialFunctions.%X52 )
      Contact( "Hmi".mainHeader[0].plcToHmi.specialFunctionButtons.active.%X40 )
      R_Coil( "Global.Data".unit[0].specialFunctions.visionUnuse )
   END_RUNG
   // the same network as SCL:
   IF "Hmi".mainHeader[0].hmiToPlc.specialFunctions.%X52 AND "Hmi".mainHeader[0].plcToHmi.specialFunctionButtons.active.%X40 THEN
       "Global.Data".unit[0].specialFunctions.visionUnuse := FALSE;
   END_IF;
END_REGION

REGION Network 13: Special Function Buttons l Run Out
   RUNG wire#powerrail
      Contact( "Hmi".mainHeader[0].plcToHmi.specialFunctionButtons.active.%X1 )
      Contact( "Hmi".mainHeader[0].plcToHmi.specialFunctionButtons.active.%X2 )
      R_Coil( "Global.Data".unit[0].specialFunctions."End of cycle" )
   END_RUNG
   // the same network as SCL:
   IF "Hmi".mainHeader[0].plcToHmi.specialFunctionButtons.active.%X1 AND "Hmi".mainHeader[0].plcToHmi.specialFunctionButtons.active.%X2 THEN
       "Global.Data".unit[0].specialFunctions."End of cycle" := FALSE;
   END_IF;
END_REGION

REGION Network 14
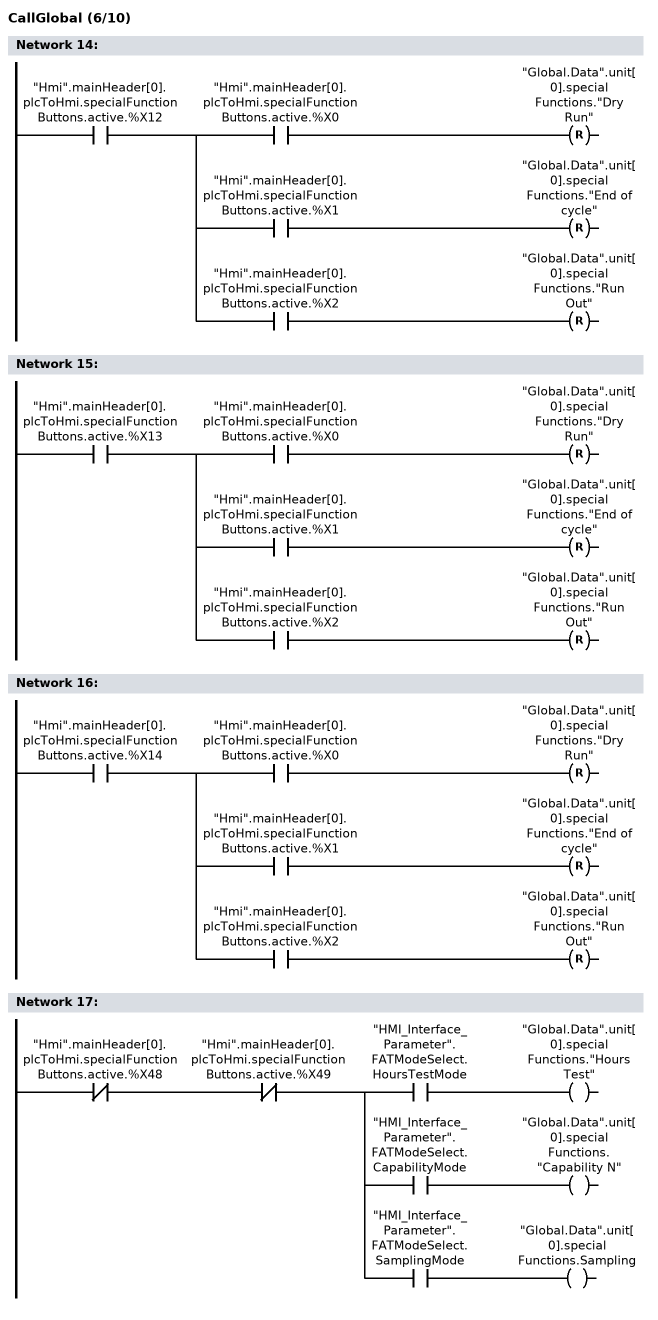
   RUNG wire#powerrail
      Contact( "Hmi".mainHeader[0].plcToHmi.specialFunctionButtons.active.%X12 )
      wire#w1
      Contact( "Hmi".mainHeader[0].plcToHmi.specialFunctionButtons.active.%X0 )
      R_Coil( "Global.Data".unit[0].specialFunctions."Dry Run" )
   END_RUNG
   RUNG wire#w1
      Contact( "Hmi".mainHeader[0].plcToHmi.specialFunctionButtons.active.%X1 )
      R_Coil( "Global.Data".unit[0].specialFunctions."End of cycle" )
   END_RUNG
   RUNG wire#w1
      Contact( "Hmi".mainHeader[0].plcToHmi.specialFunctionButtons.active.%X2 )
      R_Coil( "Global.Data".unit[0].specialFunctions."Run Out" )
   END_RUNG
   // the same network as SCL:
   IF "Hmi".mainHeader[0].plcToHmi.specialFunctionButtons.active.%X12 AND "Hmi".mainHeader[0].plcToHmi.specialFunctionButtons.active.%X0 THEN
       "Global.Data".unit[0].specialFunctions."Dry Run" := FALSE;
   END_IF;
   IF "Hmi".mainHeader[0].plcToHmi.specialFunctionButtons.active.%X12 AND "Hmi".mainHeader[0].plcToHmi.specialFunctionButtons.active.%X1 THEN
       "Global.Data".unit[0].specialFunctions."End of cycle" := FALSE;
   END_IF;
   IF "Hmi".mainHeader[0].plcToHmi.specialFunctionButtons.active.%X12 AND "Hmi".mainHeader[0].plcToHmi.specialFunctionButtons.active.%X2 THEN
       "Global.Data".unit[0].specialFunctions."Run Out" := FALSE;
   END_IF;
END_REGION

REGION Network 15
   RUNG wire#powerrail
      Contact( "Hmi".mainHeader[0].plcToHmi.specialFunctionButtons.active.%X13 )
      wire#w1
      Contact( "Hmi".mainHeader[0].plcToHmi.specialFunctionButtons.active.%X0 )
      R_Coil( "Global.Data".unit[0].specialFunctions."Dry Run" )
   END_RUNG
   RUNG wire#w1
      Contact( "Hmi".mainHeader[0].plcToHmi.specialFunctionButtons.active.%X1 )
      R_Coil( "Global.Data".unit[0].specialFunctions."End of cycle" )
   END_RUNG
   RUNG wire#w1
      Contact( "Hmi".mainHeader[0].plcToHmi.specialFunctionButtons.active.%X2 )
      R_Coil( "Global.Data".unit[0].specialFunctions."Run Out" )
   END_RUNG
   // the same network as SCL:
   IF "Hmi".mainHeader[0].plcToHmi.specialFunctionButtons.active.%X13 AND "Hmi".mainHeader[0].plcToHmi.specialFunctionButtons.active.%X0 THEN
       "Global.Data".unit[0].specialFunctions."Dry Run" := FALSE;
   END_IF;
   IF "Hmi".mainHeader[0].plcToHmi.specialFunctionButtons.active.%X13 AND "Hmi".mainHeader[0].plcToHmi.specialFunctionButtons.active.%X1 THEN
       "Global.Data".unit[0].specialFunctions."End of cycle" := FALSE;
   END_IF;
   IF "Hmi".mainHeader[0].plcToHmi.specialFunctionButtons.active.%X13 AND "Hmi".mainHeader[0].plcToHmi.specialFunctionButtons.active.%X2 THEN
       "Global.Data".unit[0].specialFunctions."Run Out" := FALSE;
   END_IF;
END_REGION

REGION Network 16
   RUNG wire#powerrail
      Contact( "Hmi".mainHeader[0].plcToHmi.specialFunctionButtons.active.%X14 )
      wire#w1
      Contact( "Hmi".mainHeader[0].plcToHmi.specialFunctionButtons.active.%X0 )
      R_Coil( "Global.Data".unit[0].specialFunctions."Dry Run" )
   END_RUNG
   RUNG wire#w1
      Contact( "Hmi".mainHeader[0].plcToHmi.specialFunctionButtons.active.%X1 )
      R_Coil( "Global.Data".unit[0].specialFunctions."End of cycle" )
   END_RUNG
   RUNG wire#w1
      Contact( "Hmi".mainHeader[0].plcToHmi.specialFunctionButtons.active.%X2 )
      R_Coil( "Global.Data".unit[0].specialFunctions."Run Out" )
   END_RUNG
   // the same network as SCL:
   IF "Hmi".mainHeader[0].plcToHmi.specialFunctionButtons.active.%X14 AND "Hmi".mainHeader[0].plcToHmi.specialFunctionButtons.active.%X0 THEN
       "Global.Data".unit[0].specialFunctions."Dry Run" := FALSE;
   END_IF;
   IF "Hmi".mainHeader[0].plcToHmi.specialFunctionButtons.active.%X14 AND "Hmi".mainHeader[0].plcToHmi.specialFunctionButtons.active.%X1 THEN
       "Global.Data".unit[0].specialFunctions."End of cycle" := FALSE;
   END_IF;
   IF "Hmi".mainHeader[0].plcToHmi.specialFunctionButtons.active.%X14 AND "Hmi".mainHeader[0].plcToHmi.specialFunctionButtons.active.%X2 THEN
       "Global.Data".unit[0].specialFunctions."Run Out" := FALSE;
   END_IF;
END_REGION

REGION Network 17
   RUNG wire#powerrail
      I_Contact( "Hmi".mainHeader[0].plcToHmi.specialFunctionButtons.active.%X48 )
      I_Contact( "Hmi".mainHeader[0].plcToHmi.specialFunctionButtons.active.%X49 )
      wire#w1
      Contact( "HMI_Interface_Parameter".FATModeSelect.HoursTestMode )
      Coil( "Global.Data".unit[0].specialFunctions."Hours Test" )
   END_RUNG
   RUNG wire#w1
      Contact( "HMI_Interface_Parameter".FATModeSelect.CapabilityMode )
      Coil( "Global.Data".unit[0].specialFunctions."Capability N" )
   END_RUNG
   RUNG wire#w1
      Contact( "HMI_Interface_Parameter".FATModeSelect.SamplingMode )
      Coil( "Global.Data".unit[0].specialFunctions.Sampling )
   END_RUNG
   // the same network as SCL:
   #_w1 := NOT "Hmi".mainHeader[0].plcToHmi.specialFunctionButtons.active.%X48 AND NOT "Hmi".mainHeader[0].plcToHmi.specialFunctionButtons.active.%X49;
   "Global.Data".unit[0].specialFunctions."Hours Test" := #_w1 AND "HMI_Interface_Parameter".FATModeSelect.HoursTestMode;
   "Global.Data".unit[0].specialFunctions."Capability N" := #_w1 AND "HMI_Interface_Parameter".FATModeSelect.CapabilityMode;
   "Global.Data".unit[0].specialFunctions.Sampling := #_w1 AND "HMI_Interface_Parameter".FATModeSelect.SamplingMode;
END_REGION

REGION Network 18: HMI Control Header
   // Read the input from the control header in the HMI an distribute information to the according units. Vice versa, summarize the unit information and provide it to the control header to display e.g. the modes and states.
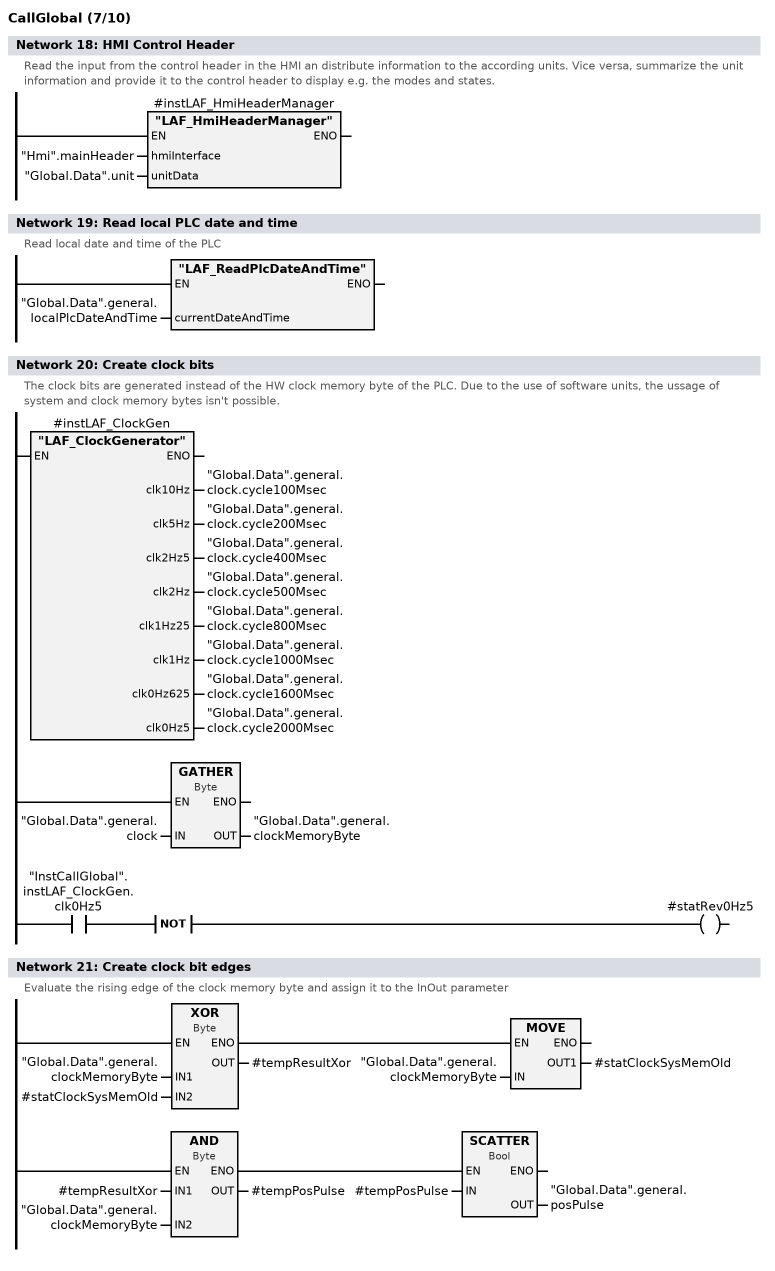
   RUNG wire#powerrail
      #instLAF_HmiHeaderManager(hmiInterface := "Hmi".mainHeader, unitData := "Global.Data".unit)
   END_RUNG
   // the same network as SCL:
   #instLAF_HmiHeaderManager(hmiInterface := "Hmi".mainHeader, unitData := "Global.Data".unit);   // "LAF_HmiHeaderManager"
END_REGION

REGION Network 19: Read local PLC date and time
   // Read local date and time of the PLC
   RUNG wire#powerrail
      "LAF_ReadPlcDateAndTime"(currentDateAndTime := "Global.Data".general.localPlcDateAndTime)
   END_RUNG
   // the same network as SCL:
   "LAF_ReadPlcDateAndTime"(currentDateAndTime := "Global.Data".general.localPlcDateAndTime);
END_REGION

REGION Network 20: Create clock bits
   // The clock bits are generated instead of the HW clock memory byte of the PLC. Due to the use of software units, the ussage of system and clock memory bytes isn't possible.
   RUNG wire#powerrail
      #instLAF_ClockGen(clk10Hz => "Global.Data".general.clock.cycle100Msec, clk5Hz => "Global.Data".general.clock.cycle200Msec, clk2Hz5 => "Global.Data".general.clock.cycle400Msec, clk2Hz => "Global.Data".general.clock.cycle500Msec, clk1Hz25 => "Global.Data".general.clock.cycle800Msec, clk1Hz => "Global.Data".general.clock.cycle1000Msec, clk0Hz625 => "Global.Data".general.clock.cycle1600Msec, clk0Hz5 => "Global.Data".general.clock.cycle2000Msec)
   END_RUNG
   RUNG wire#powerrail
      { S7_Templates := "[dest_type := Byte, src_type := Bool]" } GATHER(IN := "Global.Data".general.clock, OUT => "Global.Data".general.clockMemoryByte)
   END_RUNG
   RUNG wire#powerrail
      Contact( "InstCallGlobal".instLAF_ClockGen.clk0Hz5 )
      Not()
      Coil( #statRev0Hz5 )
   END_RUNG
   // the same network as SCL:
   #instLAF_ClockGen(clk10Hz => "Global.Data".general.clock.cycle100Msec,   // "LAF_ClockGenerator"
                     clk5Hz => "Global.Data".general.clock.cycle200Msec,
                     clk2Hz5 => "Global.Data".general.clock.cycle400Msec,
                     clk2Hz => "Global.Data".general.clock.cycle500Msec,
                     clk1Hz25 => "Global.Data".general.clock.cycle800Msec,
                     clk1Hz => "Global.Data".general.clock.cycle1000Msec,
                     clk0Hz625 => "Global.Data".general.clock.cycle1600Msec,
                     clk0Hz5 => "Global.Data".general.clock.cycle2000Msec);
   GATHER(IN := "Global.Data".general.clock, OUT => "Global.Data".general.clockMemoryByte);
   #statRev0Hz5 := NOT "InstCallGlobal".instLAF_ClockGen.clk0Hz5;
END_REGION

REGION Network 21: Create clock bit edges
   // Evaluate the rising edge of the clock memory byte and assign it to the InOut parameter
   #tempResultXor := "Global.Data".general.clockMemoryByte XOR #statClockSysMemOld;
   #statClockSysMemOld := "Global.Data".general.clockMemoryByte;
   #tempPosPulse := #tempResultXor AND "Global.Data".general.clockMemoryByte;
   SCATTER(IN := #tempPosPulse, OUT => "Global.Data".general.posPulse);
END_REGION

REGION Network 22: Time Synchronisation (NTP)
   // With the LSNTP_Server block, the NTP server will be enabled on S7 PLC, to wich the NTP client (e.g. Panel), can synchronize their data and time.
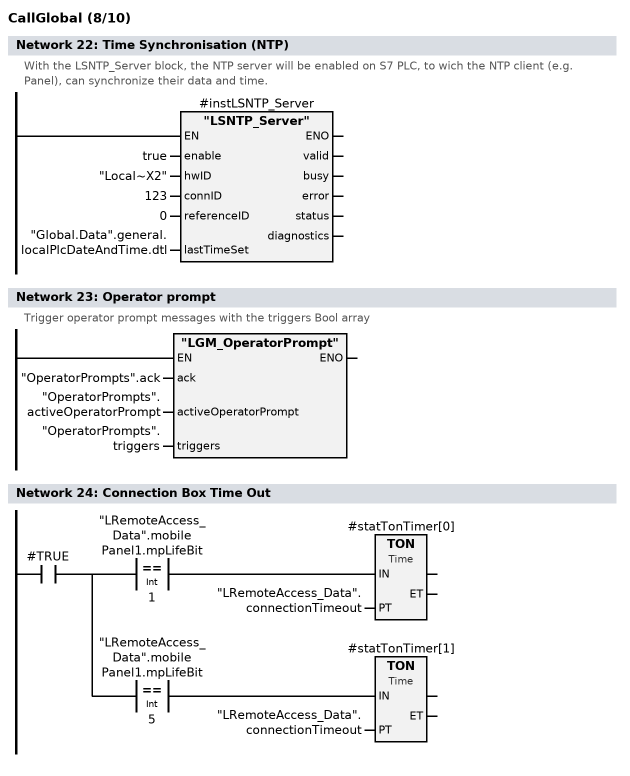
   RUNG wire#powerrail
      #instLSNTP_Server(enable := true, hwID := "Local~X2", connID := 123, referenceID := 0, lastTimeSet := "Global.Data".general.localPlcDateAndTime.dtl, valid =>, busy =>, error =>, status =>, diagnostics =>)
   END_RUNG
   // the same network as SCL:
   #instLSNTP_Server(enable := true,   // "LSNTP_Server"
                     hwID := "Local~X2",
                     connID := 123,
                     referenceID := 0,
                     lastTimeSet := "Global.Data".general.localPlcDateAndTime.dtl);
END_REGION

REGION Network 23: Operator prompt
   // Trigger operator prompt messages with the triggers Bool array
   RUNG wire#powerrail
      "LGM_OperatorPrompt"(ack := "OperatorPrompts".ack, activeOperatorPrompt := "OperatorPrompts".activeOperatorPrompt, triggers := "OperatorPrompts".triggers)
   END_RUNG
   // the same network as SCL:
   "LGM_OperatorPrompt"(ack := "OperatorPrompts".ack,
                        activeOperatorPrompt := "OperatorPrompts".activeOperatorPrompt,
                        triggers := "OperatorPrompts".triggers);
END_REGION

REGION Network 24: Connection Box Time Out
   RUNG wire#powerrail
      Contact( #TRUE )
      wire#w1
      { S7_Templates := "SrcType := Int" } EQ_Contact(in1 := "LRemoteAccess_Data".mobilePanel1.mpLifeBit, in2 := 1)
      { S7_Templates := "time_type := Time" } #statTonTimer[0].TON(pt := "LRemoteAccess_Data".connectionTimeout, et =>)
   END_RUNG
   RUNG wire#w1
      { S7_Templates := "SrcType := Int" } EQ_Contact(in1 := "LRemoteAccess_Data".mobilePanel1.mpLifeBit, in2 := 5)
      { S7_Templates := "time_type := Time" } #statTonTimer[1].TON(pt := "LRemoteAccess_Data".connectionTimeout, et =>)
   END_RUNG
   // the same network as SCL:
   #statTonTimer[0].TON(IN := #TRUE AND ("LRemoteAccess_Data".mobilePanel1.mpLifeBit = 1),
                        PT := "LRemoteAccess_Data".connectionTimeout);
   #statTonTimer[1].TON(IN := #TRUE AND ("LRemoteAccess_Data".mobilePanel1.mpLifeBit = 5),
                        PT := "LRemoteAccess_Data".connectionTimeout);
END_REGION

REGION Network 25: Connection box is connected
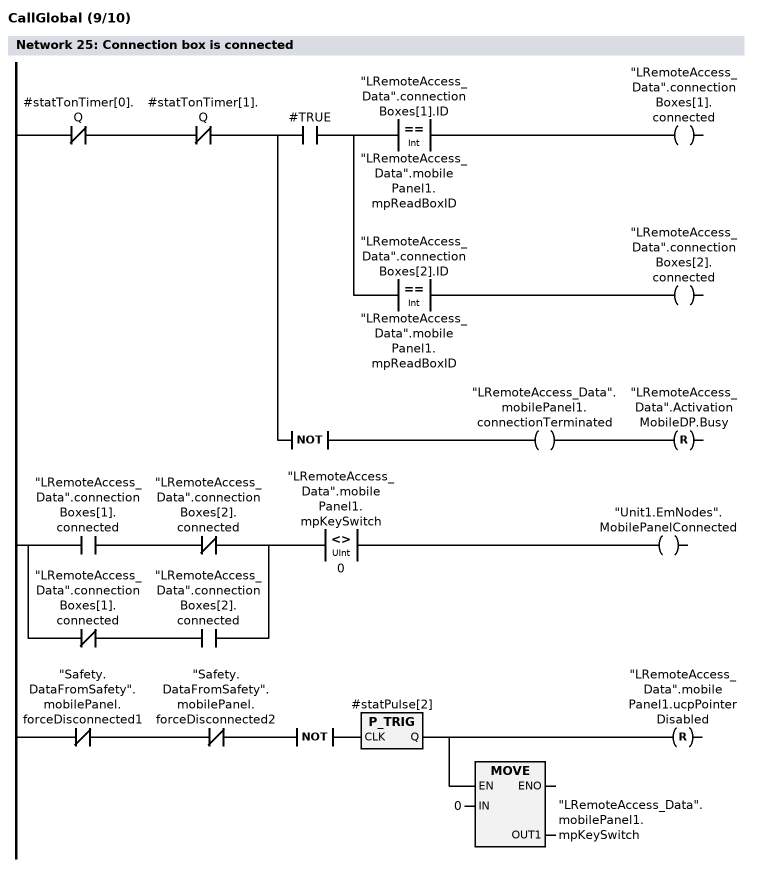
   RUNG wire#powerrail
      I_Contact( #statTonTimer[0].Q )
      I_Contact( #statTonTimer[1].Q )
      wire#w1
      Contact( #TRUE )
      wire#w2
      { S7_Templates := "SrcType := Int" } EQ_Contact(in1 := "LRemoteAccess_Data".connectionBoxes[1].ID, in2 := "LRemoteAccess_Data".mobilePanel1.mpReadBoxID)
      Coil( "LRemoteAccess_Data".connectionBoxes[1].connected )
   END_RUNG
   RUNG wire#w2
      { S7_Templates := "SrcType := Int" } EQ_Contact(in1 := "LRemoteAccess_Data".connectionBoxes[2].ID, in2 := "LRemoteAccess_Data".mobilePanel1.mpReadBoxID)
      Coil( "LRemoteAccess_Data".connectionBoxes[2].connected )
   END_RUNG
   RUNG wire#w1
      Not()
      Coil( "LRemoteAccess_Data".mobilePanel1.connectionTerminated )
      R_Coil( "LRemoteAccess_Data".ActivationMobileDP.Busy )
   END_RUNG
   RUNG wire#powerrail
      Contact( "LRemoteAccess_Data".connectionBoxes[1].connected )
      I_Contact( "LRemoteAccess_Data".connectionBoxes[2].connected )
      wire#w3
      { S7_Templates := "SrcType := UInt" } NE_Contact(in1 := "LRemoteAccess_Data".mobilePanel1.mpKeySwitch, in2 := 0)
      Coil( "Unit1.EmNodes".MobilePanelConnected )
   END_RUNG
   RUNG wire#powerrail
      I_Contact( "LRemoteAccess_Data".connectionBoxes[1].connected )
      Contact( "LRemoteAccess_Data".connectionBoxes[2].connected )
   END_RUNG wire#w3
   RUNG wire#powerrail
      I_Contact( "Safety.DataFromSafety".mobilePanel.forceDisconnected1 )
      I_Contact( "Safety.DataFromSafety".mobilePanel.forceDisconnected2 )
      Not()
      P_Trig( #statPulse[2] )
      wire#w4
      R_Coil( "LRemoteAccess_Data".mobilePanel1.ucpPointerDisabled )
   END_RUNG
   RUNG wire#w4
      Move(in := 0, out1 => "LRemoteAccess_Data".mobilePanel1.mpKeySwitch)
   END_RUNG
   // the same network as SCL:
   #_w1 := NOT #statTonTimer[0].Q AND NOT #statTonTimer[1].Q;
   #_w2 := #_w1 AND #TRUE;
   "LRemoteAccess_Data".connectionBoxes[1].connected := #_w2 AND ("LRemoteAccess_Data".connectionBoxes[1].ID = "LRemoteAccess_Data".mobilePanel1.mpReadBoxID);
   "LRemoteAccess_Data".connectionBoxes[2].connected := #_w2 AND ("LRemoteAccess_Data".connectionBoxes[2].ID = "LRemoteAccess_Data".mobilePanel1.mpReadBoxID);
   "LRemoteAccess_Data".mobilePanel1.connectionTerminated := NOT #_w1;
   IF NOT #_w1 THEN "LRemoteAccess_Data".ActivationMobileDP.Busy := FALSE; END_IF;
   "Unit1.EmNodes".MobilePanelConnected := (("LRemoteAccess_Data".connectionBoxes[1].connected AND NOT "LRemoteAccess_Data".connectionBoxes[2].connected) OR (NOT "LRemoteAccess_Data".connectionBoxes[1].connected AND "LRemoteAccess_Data".connectionBoxes[2].connected)) AND ("LRemoteAccess_Data".mobilePanel1.mpKeySwitch <> 0);
   #_w3 := NOT (NOT "Safety.DataFromSafety".mobilePanel.forceDisconnected1 AND NOT "Safety.DataFromSafety".mobilePanel.forceDisconnected2);
   #_w4 := #_w3 AND NOT #statPulse[2];   // rising edge
   #statPulse[2] := #_w3;
   IF #_w4 THEN
       "LRemoteAccess_Data".mobilePanel1.ucpPointerDisabled := FALSE;
       "LRemoteAccess_Data".mobilePanel1.mpKeySwitch := 0;
   END_IF;
END_REGION

REGION Network 26: LRemoteAccess_Data → DataToSafety
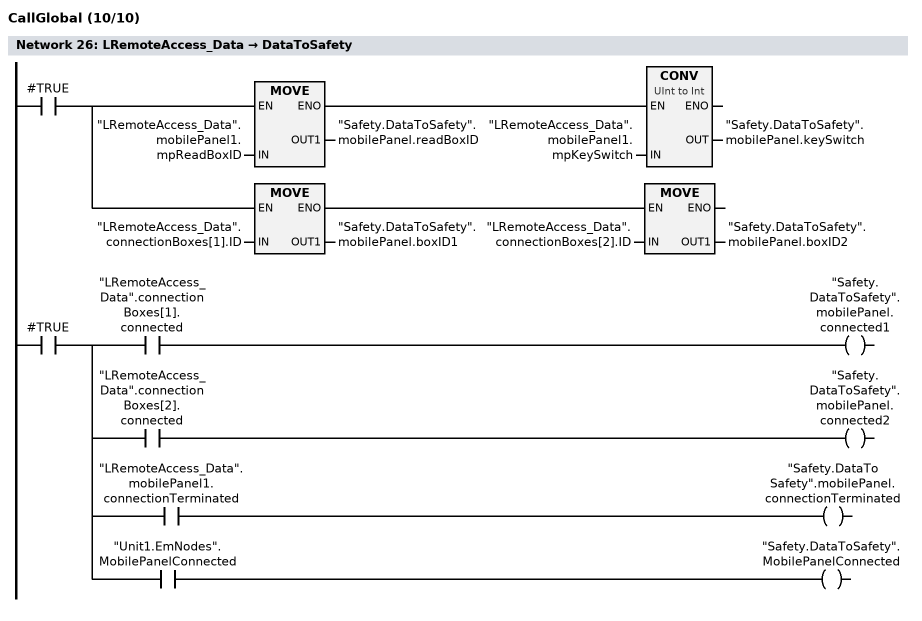
   RUNG wire#powerrail
      Contact( #TRUE )
      wire#w1
      Move(in := "LRemoteAccess_Data".mobilePanel1.mpReadBoxID, out1 => "Safety.DataToSafety".mobilePanel.readBoxID)
      { S7_Templates := "[SrcType := UInt, DestType := Int]" } Convert(in := "LRemoteAccess_Data".mobilePanel1.mpKeySwitch, out => "Safety.DataToSafety".mobilePanel.keySwitch)
   END_RUNG
   RUNG wire#w1
      Move(in := "LRemoteAccess_Data".connectionBoxes[1].ID, out1 => "Safety.DataToSafety".mobilePanel.boxID1)
      Move(in := "LRemoteAccess_Data".connectionBoxes[2].ID, out1 => "Safety.DataToSafety".mobilePanel.boxID2)
   END_RUNG
   RUNG wire#powerrail
      Contact( #TRUE )
      wire#w2
      Contact( "LRemoteAccess_Data".connectionBoxes[1].connected )
      Coil( "Safety.DataToSafety".mobilePanel.connected1 )
   END_RUNG
   RUNG wire#w2
      Contact( "LRemoteAccess_Data".connectionBoxes[2].connected )
      Coil( "Safety.DataToSafety".mobilePanel.connected2 )
   END_RUNG
   RUNG wire#w2
      Contact( "LRemoteAccess_Data".mobilePanel1.connectionTerminated )
      Coil( "Safety.DataToSafety".mobilePanel.connectionTerminated )
   END_RUNG
   RUNG wire#w2
      Contact( "Unit1.EmNodes".MobilePanelConnected )
      Coil( "Safety.DataToSafety".MobilePanelConnected )
   END_RUNG
   // the same network as SCL:
   IF #TRUE THEN
       "Safety.DataToSafety".mobilePanel.readBoxID := "LRemoteAccess_Data".mobilePanel1.mpReadBoxID;
       "Safety.DataToSafety".mobilePanel.keySwitch := UINT_TO_INT("LRemoteAccess_Data".mobilePanel1.mpKeySwitch);
       "Safety.DataToSafety".mobilePanel.boxID1 := "LRemoteAccess_Data".connectionBoxes[1].ID;
       "Safety.DataToSafety".mobilePanel.boxID2 := "LRemoteAccess_Data".connectionBoxes[2].ID;
   END_IF;
   "Safety.DataToSafety".mobilePanel.connected1 := #TRUE AND "LRemoteAccess_Data".connectionBoxes[1].connected;
   "Safety.DataToSafety".mobilePanel.connected2 := #TRUE AND "LRemoteAccess_Data".connectionBoxes[2].connected;
   "Safety.DataToSafety".mobilePanel.connectionTerminated := #TRUE AND "LRemoteAccess_Data".mobilePanel1.connectionTerminated;
   "Safety.DataToSafety".MobilePanelConnected := #TRUE AND "Unit1.EmNodes".MobilePanelConnected;
END_REGION
END_FUNCTION_BLOCK
